// TIA Portal V16 export
// export: Created 2019-09-22T11:06:18.4384038Z, ExportSetting WithDefaults, DisplayName Totally Integrated Automation Portal, DisplayVersion V16, DisplayName TIA Portal Version Control Interface, DisplayVersion V16, DisplayName TIA Portal Openness, DisplayVersion V16, DisplayName STEP 7 Professional, DisplayVersion V16, DisplayName SIMATIC Energy Suite, DisplayVersion V16, DisplayName STEP 7 Safety, DisplayVersion V16, DisplayName WinCC Professional, DisplayVersion V16, DisplayName SIMATIC Visualization Architect, DisplayVersion V16
DATA_BLOCK "InstDiagnostics"   // DB2000
VERSION : 0.1
// stored: AutoNumber true, InstanceOfName Diagnostics, InstanceOfType FB
"Diagnostics"
   // VAR_INPUT
   //    firstCyleInit : Bool;
   // END_VAR
   // VAR_IN_OUT
   //    plc : "typePlc";
   //    showPlc : "typeShowPlc";
   //    ioSystem : Array[1.."MAX_SYSTEM"] of "typeIoSystem";
   //    showIoSystem : Array[1.."MAX_SYSTEM"] of "typeShowIoSystem";
   //    showActIoSystem : "typeShowActIoSystem";
   // END_VAR
   // VAR
   //    statIoSystemIndex : Int;
   //    statSlotIndex : Int;
   //    statDeviceIndex : Int;
   // END_VAR
BEGIN
END_DATA_BLOCK
